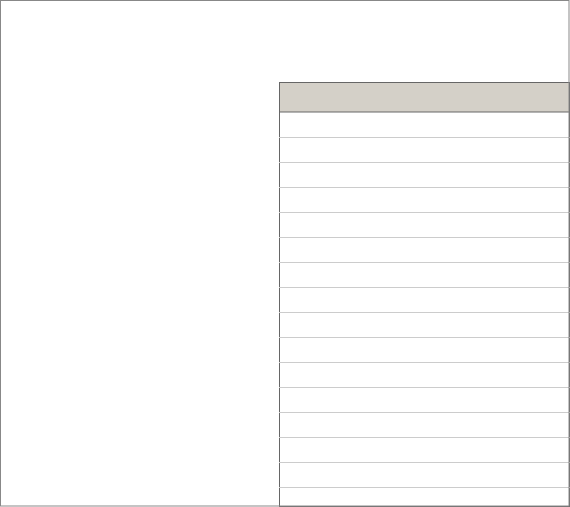
VISUALIZATION Visualization_ThermostaatTijdsturing  // 570x507
    Table (279,82 291x425), data array: prg_ThermostaatregelingTijdsturing.TempLog
        p3854506369: prg_ThermostaatregelingTijdsturing.TempLog[INDEX]
        p2232123230: Temperatuur
        Columns.Column.[0].Template: prg_ThermostaatregelingTijdsturing.TempAlarm
END_VISUALIZATION

(* stored: Version 1.1.0.1, ProductVersion 3.1.4024.15
   Visu Visualization_ThermostaatTijdsturing: Id {7d2f36d8-70fa-4514-a2b5-e2251fbb23b9} *)
